{region '#Template'}
	{attribute 'Version' := '5.0.0.0'}
	{attribute 'Tags' := '"LCID": "1031", "Text": "Trade, Plant, Heating System"'}
	{attribute 'Tags' := '"LCID": "1033", "Text": "Trade, Plant, Heating System"'}
	{attribute 'Using' := '"Type": "Template", "URI": "Site"'}
	{attribute 'Description' := '"LCID": "1031", "Text": "Aufruf der Anlagen des Gewerks Heizsysteme"'}
	{attribute 'Description' := '"LCID": "1033", "Text": "Calling the plants of the trade heating system"'}
{endregion}
FUNCTION_BLOCK FB_BA_Heating EXTENDS FB_BA_View
VAR_INPUT CONSTANT
	HTC01				: FB_BA_H_HtgCir01;		
END_VAR
VAR_INPUT
END_VAR
VAR_OUTPUT
END_VAR
VAR
END_VAR

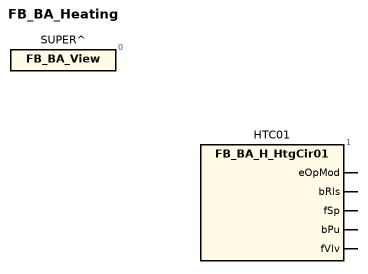
SUPER^(); // FB_BA_View
HTC01(); // FB_BA_H_HtgCir01

METHOD FB_init : BOOL
VAR_INPUT
	bInitRetains : BOOL; // if TRUE, the retain variables are initialized (warm start / cold start)
	bInCopyCode : BOOL;  // if TRUE, the instance afterwards gets moved into the copy code (online change)
END_VAR
HTC01.iParent 					:= THIS^;	
HTC01.iLabel						:= LblPlt_Heating_circuit;	
HTC01.sObjectName					:= '{Idx=01}';          
HTC01.eDPADMode					:= E_BA_DPADMode.eInclude;
END_METHOD

END_FUNCTION_BLOCK

(* stored: Version 1.1.0.1, ProductVersion 3.1.4024.12
   POU FB_BA_Heating: Id {90f3b4c6-089f-49c4-a972-6fac0971f9b6}, SpecialFunc None
   Method FB_init: Id {aa91cbcf-a991-41d7-bcac-620d9975e82e} *)
